TYPE TcoLiftingRotaryTransfer_Status EXTENDS TcoCore.TcoStruct:
STRUCT


		ActionDescription:STRING;
		
END_STRUCT
END_TYPE

(* stored: Version 1.1.0.1
   DUT TcoLiftingRotaryTransfer_Status: Id {8607e361-bfa6-4bca-9098-00584a439579} *)
